# EPICS StreamDevice protocol: Tektronix_MSO58LPSup/devTektronix_MSO58LP.proto
OutTerminator = '\n';
ReplyTimeout = 1500;

getIDN {
    out "*IDN?";
    #Read no more that 39 chars (EPICS limit)
    in "%/(.{0,39})/";
    ExtraInput = Ignore;
}

readIDNParts {
    out "*IDN?";
    in "%(\$1)[_a-zA-Z0-9],%(\$2)[_a-zA-Z0-9],%(\$3)[_a-zA-Z0-9],CF:%(\$4)[a-zA-Z0-9\.] FV:%(\$5)[_a-zA-Z0-9\.]";
	ExtraInput = Ignore;

}

getXINC {
	#get x increment for plot
	out ":DATa:SOUrce CH\$1";
	wait 10;
	out "WFMOutpre:XINcr?";
	in "%f";
	ExtraInput = Ignore;
}

getYMULT {
	#get y multiplier for plot
	out ":DATa:SOUrce CH\$1";
	wait 10;
	out "WFMOutpre:YMUlt?";
	in "%f";
	ExtraInput = Ignore;
}

getXUNIT {
	#get x unit for plot
	out ":DATa:SOUrce CH\$1";
	wait 10;
	out "WFMOutpre:XUNit?";
	in '%/([a-zA-Z]+)/';
	ExtraInput = Ignore;
}

getYUNIT {
	#get y unit for plot
	out ":DATa:SOUrce CH\$1";
	wait 10;
	out "WFMOutpre:YUNit?";
	in '%/([a-zA-Z]+)/';
	ExtraInput = Ignore;
}

getYDATA {
	#ask scope for y data points
	out ":VERBOSE 0";
	wait 1;
	out "HEADER 0";
	wait 1;
	out ":DATa:SOUrce CH\$1";
	wait 1;
	out ":DATa:STARt 1";
	wait 1;
	out ":DATa:STOP \$2";
	wait 1;
	out ":DATa:ENCdg ASCIi";
	wait 1;
	out ":DATa:WIDth 1";
	wait 1;
	out ":CURVe?";
	separator=",";
	in "%d";
	ExtraInput = Ignore;
}
